Universal Robots PolyScope program: push_motor_plate.urp

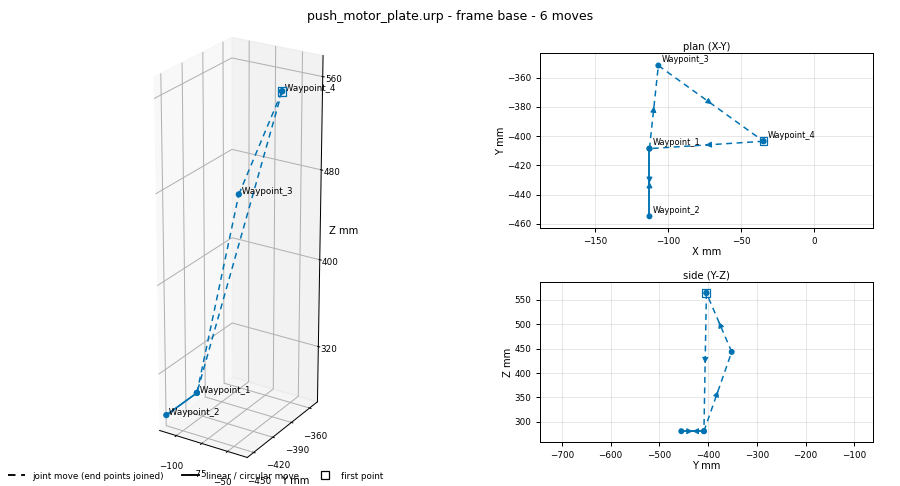
[picture p0: tool path of push_motor_plate.urp in frame base, 6 of 7 moves have a stored position in this frame; points joined in program order, loops and branches not executed]
Program wrs2020_push_motor_plate (installation=default directory=/programs createdIn=5.7.0.90932 lastSavedIn=5.7.0.90932 robotSerialNumber=20205500607)
Calibrated DH parameters: a=[0.000096, -0.337, -0.383372, 0.000118, 0.000015, 0]; d=[0.162724, 79.377998, -95.545185, 16.300583, 0.099689, 0.099499]; alpha=[1.569249, 0.003272, 0.005201, 1.570041, -1.570219, 0]; deltaTheta=[0, 0.65664, 5.410619, 0.215927, -0.000001, 0]
Robot Program (runOnlyOnce=true)
  Set NoAction tcp=TCP
  pose0 := get_actual_tcp_pose()
  URCap Gripper (Robotiq_Grippers, Robotiq Inc.) dataModel(position=100.0, force=0.0, speed=100.0, positionInDouble=100.0, forceInDouble=0.0, speedInDouble=100.0, slaveIds=[9], blocking=true)
  MoveJ speed 60 deg/s, acceleration 80 deg/s^2 (useActiveTCP=false) tcp=TCP; feature=Base
    Waypoint Waypoint_4: TCP in base x=-34.781 y=-403.495 z=564.378 mm, rx=1.6505 ry=-1.5845 rz=-0.8753 rad; joints [77.92, -104.184, 102.705, -108.391, -144.334, -114.84] deg
  MoveJ speed 60 deg/s, acceleration 80 deg/s^2 (useActiveTCP=false) tcp=TCP; feature=Base
    Waypoint Waypoint_1: TCP in base x=-112.977 y=-408.527 z=280.885 mm, rx=1.9666 ry=-2.0326 rz=0.4017 rad; joints [53.141, -95.017, 133.793, -147.812, -76.696, -122.667] deg
  MoveL speed 250 mm/s, acceleration 1200 mm/s^2 (useActiveTCP=false) tcp=TCP; feature=Base
    Waypoint Waypoint_2: motionParameters(jointSpeed=1.047198 jointAcceleration=1.396263 cartesianSpeed=0.01 cartesianAcceleration=1.2); TCP in base x=-112.977 y=-454.965 z=280.885 mm, rx=1.9666 ry=-2.0326 rz=0.4017 rad; joints [57.073, -88.288, 127.58, -149.144, -77.997, -118.846] deg
    Wait Sleep waitTime=0.5
    Waypoint Waypoint_1: TCP in base x=-112.977 y=-408.527 z=280.885 mm, rx=1.9666 ry=-2.0326 rz=0.4017 rad; joints [53.141, -95.017, 133.793, -147.812, -76.696, -122.667] deg
  MoveJ speed 60 deg/s, acceleration 80 deg/s^2 (useActiveTCP=false) tcp=TCP; feature=Base
    Waypoint Waypoint_3: TCP in base x=-106.875 y=-351.582 z=443.459 mm, rx=1.8757 ry=-1.5471 rz=-0.3518 rad; joints [57.352, -112.494, 127.33, -143.483, -108.632, -140.235] deg
  URCap Gripper (Robotiq_Grippers, Robotiq Inc.) dataModel(position=0.0, force=0.0, speed=100.0, positionInDouble=0.0, forceInDouble=0.0, speedInDouble=100.0, slaveIds=[9], blocking=true)
  MoveJ speed 60 deg/s, acceleration 80 deg/s^2 (useActiveTCP=false) tcp=TCP; feature=Base
    Waypoint Waypoint_4: TCP in base x=-34.781 y=-403.495 z=564.378 mm, rx=1.6505 ry=-1.5845 rz=-0.8753 rad; joints [77.92, -104.184, 102.705, -108.391, -144.334, -114.84] deg
    Waypoint Waypoint_5 (Variable): variable=pose0
